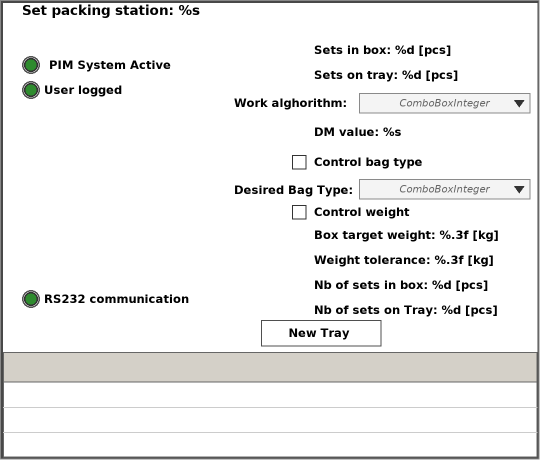
VISUALIZATION vSetPacking_Status  // 540x460
VAR_IN_OUT
	fbData:fbSetPackingStation_V3;
END_VAR
    Rectangle (1,1 538x458), "Set packing station: %s", text variable: fbData.stStationData.sNazwaStanowiska
    RoundedRectangle (18,55 193x20), "PIM System Active", colour toggle: NOT fbData.bPIM_Active
    Label (41,80 170x20), "User logged"
    Lamp1 (21,80 20x20), variable: fbData.bUserLogged, style: Lamp-Lamp1-Green
    Lamp1 (21,289 20x20), variable: fbData.bCommRS232Axis_OK, style: Lamp-Lamp1-Green
    Label (41,289 170x20), "RS232 communication"
    Lamp1 (21,55 20x20), variable: fbData.bPIM_Active, style: Lamp-Lamp1-Green
    Rectangle (311,65 200x20), "Sets on tray: %d [pcs]", text variable: fbData.iNbOfSetsOnTray, input disabled if: NOT GVL.fbUserLogin.bPermissionGranted
        OnMouseClick: write the text variable via Default, min 0, max 1000
    Rectangle (311,122 200x20), "DM value: %s", text variable: fbData.stTestData.sDataMatrixText, input disabled if: NOT GVL.fbUserLogin.bPermissionGranted
        OnMouseClick: write the text variable via Edit, title 'DM value'
    Rectangle (311,225 200x20), "Box target weight: %.3f [kg]", text variable: fbData.stTestData.rTargetWeight, input disabled if: NOT GVL.fbUserLogin.bPermissionGranted
        OnMouseClick: write fbData.stTestData.rTargetWeight via Default, min 0.5, max 20, title 'Box weight', format %.1f
    Rectangle (311,250 200x20), "Weight tolerance: %.3f [kg]", text variable: fbData.stTestData.rMaxWeightDeviation, input disabled if: NOT GVL.fbUserLogin.bPermissionGranted
        OnMouseClick: write fbData.stTestData.rMaxWeightDeviation via Default, min 0.01, max 2.0, title 'Weight tolerance', format %.1f
    Rectangle (311,275 200x20), "Nb of sets in box: %d [pcs]", text variable: fbData.stTestData.iNumberOfSetsInBox, input disabled if: NOT GVL.fbUserLogin.bPermissionGranted
        OnMouseClick: write the text variable via Default, min 1, max 100, title 'Nb of sets in box', format %d
    Rectangle (311,300 200x20), "Nb of sets on Tray: %d [pcs]", text variable: fbData.stTestData.iNumberOfSetsOnTray, input disabled if: NOT GVL.fbUserLogin.bPermissionGranted
        OnMouseClick: write the text variable via Default, min 0, max 1000
    Rectangle (311,40 200x20), "Sets in box: %d [pcs]", text variable: fbData.iSetsInBufferCtr
        OnMouseClick: write the text variable via Default, min 0, max (fbData.stTestData.iNumberOfSetsInBox-1), format %d
    Rectangle (261,320 120x26), "New Tray", colour toggle: fbData.bNewTray, input disabled if: Not GVL.fbUserLogin.bPermissionGranted
    Table (3,352 534x105), data array: fbData.fbAlarmTab.astErrTable
        p1128707560: fbData.fbAlarmTab.uiRowNumber
        p3854506369: fbData.fbAlarmTab.astErrTable[INDEX].dtEventTime
        p1892666644: fbData.fbAlarmTab.astErrTable[INDEX].sMachineId
        p338671338: fbData.fbAlarmTab.astErrTable[INDEX].sEventDescription
        p2170511999: fbData.fbAlarmTab.astErrTable[INDEX].dwErrorCode
        p3723444502: fbData.fbAlarmTab.astErrTable[INDEX].uiRepeatQty
        p1218418051: fbData.fbAlarmTab.astErrTable[INDEX].nAlarmClass
        p4092479075: Error Code
        p2237128397: Repeat Qty
    Checkbox (290,202 20x20), variable: fbData.stTestData.bControlWeight, input disabled if: NOT GVL.fbUserLogin.bPermissionGranted
    Label (311,202 170x20), "Control weight"
    ComboBoxInteger (359,93 171x20), variable: fbData.stTestData.nWorkAlgorithm, input disabled if: NOT GVL.fbUserLogin.bPermissionGranted
    Label (231,93 128x20), "Work alghorithm:"
    Rectangle (231,180 132x20), "Desired Bag Type:", input disabled if: NOT GVL.fbUserLogin.bPermissionGranted
    Checkbox (290,152 20x20), variable: fbData.stTestData.bCheckBagType, input disabled if: NOT GVL.fbUserLogin.bPermissionGranted
    Label (311,152 170x20), "Control bag type"
    ComboBoxInteger (359,179 171x20), variable: fbData.stTestData.nDesiredBagType, input disabled if: NOT GVL.fbUserLogin.bPermissionGranted
END_VISUALIZATION

(* stored: Version 1.1.0.1, ProductVersion 3.1.4024.12
   Visu vSetPacking_Status: Id {697088b0-1bcd-4b90-8b18-d8da68b6e8c3} *)
